// TIA Portal project "CAFERSERHAT_YAĞCI_TMR08" (V14)

(* hardware
DEVICE "S7-1200 station_1"  S7-1200 Station
   slot 0: "Rack_0"  Rack  V1.0
   slot 1: "PLC_1"  CPU 1214C DC/DC/DC  6ES7 214-1AG40-0XB0  V4.1
*)

// ===== PLC "PLC_1"  CPU 1214C DC/DC/DC =====

VAR_GLOBAL   // PLC tag table "GİRİŞ VE ÇIKIŞ ETİKETLERİ"
   "S1 NK" AT %I0.0 : Bool;
   "S5 NA" AT %I0.1 : Bool;
   "S8 NA" AT %I0.2 : Bool;
   "S8 NK" AT %I0.3 : Bool;
   "S2 NA" AT %I0.4 : Bool;
   "S2 NK" AT %I0.5 : Bool;
   "S3 NK" AT %I0.6 : Bool;
   "S3 NA" AT %I0.7 : Bool;
   "S4 NK" AT %I1.0 : Bool;
   "S4 NA" AT %I1.1 : Bool;
   "S7 NA" AT %I1.2 : Bool;
   "S7 NK" AT %I1.3 : Bool;
   "S6 NK" AT %I1.4 : Bool;
   "S6 NA" AT %I1.5 : Bool;
   "Tag_15" AT %I1.6 : Bool;
   "H2 SARI LAMBA" AT %Q0.0 : Bool;
   "H1 KIRMIZI LAMBA" AT %Q0.1 : Bool;
   "H3 SARI LAMBA" AT %Q0.2 : Bool;
   "H6 SARI LAMBA" AT %Q0.3 : Bool;
   "H5 YEŞİL LAMBA" AT %Q0.4 : Bool;
   "H7 MAVİ LAMBA" AT %Q0.5 : Bool;
   "Tag_22" AT %Q0.6 : Bool;
   "H4 YEŞİL LAMBA" AT %Q0.7 : Bool;
   "Tag_24" AT %Q1.0 : Bool;
   "Tag_25" AT %Q1.1 : Bool;
END_VAR

ORGANIZATION_BLOCK "SORU 1"   // OB1, LAD, ProgramCycle
TITLE = "Main Program Sweep (Cycle)"
{ S7_Optimized_Access := 'TRUE' }
VERSION : 0.1
   VAR_INPUT
      Initial_Call : Bool;   // Initial call of this OB
      Remanence : Bool;   // =True, if remanent data are available
   END_VAR
BEGIN

REGION Network 1
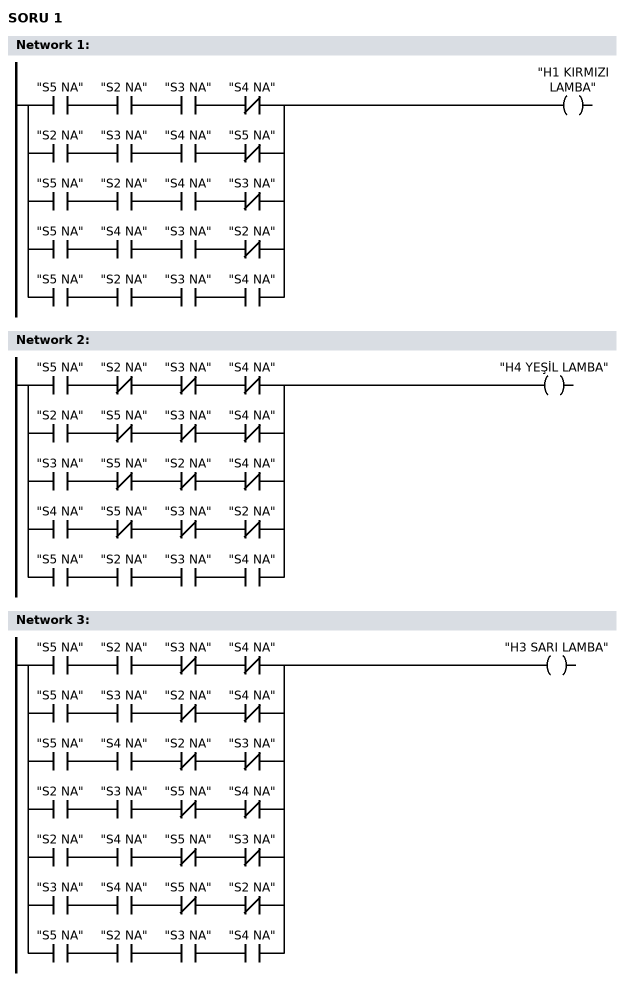
   RUNG wire#powerrail
      Contact( "S5 NA" )
      Contact( "S2 NA" )
      Contact( "S3 NA" )
      I_Contact( "S4 NA" )
      wire#w1
      Coil( "H1 KIRMIZI LAMBA" )
   END_RUNG
   RUNG wire#powerrail
      Contact( "S2 NA" )
      Contact( "S3 NA" )
      Contact( "S4 NA" )
      I_Contact( "S5 NA" )
   END_RUNG wire#w1
   RUNG wire#powerrail
      Contact( "S5 NA" )
      Contact( "S2 NA" )
      Contact( "S4 NA" )
      I_Contact( "S3 NA" )
   END_RUNG wire#w1
   RUNG wire#powerrail
      Contact( "S5 NA" )
      Contact( "S4 NA" )
      Contact( "S3 NA" )
      I_Contact( "S2 NA" )
   END_RUNG wire#w1
   RUNG wire#powerrail
      Contact( "S5 NA" )
      Contact( "S2 NA" )
      Contact( "S3 NA" )
      Contact( "S4 NA" )
   END_RUNG wire#w1
   // the same network as SCL:
   "H1 KIRMIZI LAMBA" := ("S5 NA" AND "S2 NA" AND "S3 NA" AND NOT "S4 NA") OR ("S2 NA" AND "S3 NA" AND "S4 NA" AND NOT "S5 NA") OR ("S5 NA" AND "S2 NA" AND "S4 NA" AND NOT "S3 NA") OR ("S5 NA" AND "S4 NA" AND "S3 NA" AND NOT "S2 NA") OR ("S5 NA" AND "S2 NA" AND "S3 NA" AND "S4 NA");
END_REGION

REGION Network 2
   RUNG wire#powerrail
      Contact( "S5 NA" )
      I_Contact( "S2 NA" )
      I_Contact( "S3 NA" )
      I_Contact( "S4 NA" )
      wire#w1
      Coil( "H4 YEŞİL LAMBA" )
   END_RUNG
   RUNG wire#powerrail
      Contact( "S2 NA" )
      I_Contact( "S5 NA" )
      I_Contact( "S3 NA" )
      I_Contact( "S4 NA" )
   END_RUNG wire#w1
   RUNG wire#powerrail
      Contact( "S3 NA" )
      I_Contact( "S5 NA" )
      I_Contact( "S2 NA" )
      I_Contact( "S4 NA" )
   END_RUNG wire#w1
   RUNG wire#powerrail
      Contact( "S4 NA" )
      I_Contact( "S5 NA" )
      I_Contact( "S3 NA" )
      I_Contact( "S2 NA" )
   END_RUNG wire#w1
   RUNG wire#powerrail
      Contact( "S5 NA" )
      Contact( "S2 NA" )
      Contact( "S3 NA" )
      Contact( "S4 NA" )
   END_RUNG wire#w1
   // the same network as SCL:
   "H4 YEŞİL LAMBA" := ("S5 NA" AND NOT "S2 NA" AND NOT "S3 NA" AND NOT "S4 NA") OR ("S2 NA" AND NOT "S5 NA" AND NOT "S3 NA" AND NOT "S4 NA") OR ("S3 NA" AND NOT "S5 NA" AND NOT "S2 NA" AND NOT "S4 NA") OR ("S4 NA" AND NOT "S5 NA" AND NOT "S3 NA" AND NOT "S2 NA") OR ("S5 NA" AND "S2 NA" AND "S3 NA" AND "S4 NA");
END_REGION

REGION Network 3
   RUNG wire#powerrail
      Contact( "S5 NA" )
      Contact( "S2 NA" )
      I_Contact( "S3 NA" )
      I_Contact( "S4 NA" )
      wire#w1
      Coil( "H3 SARI LAMBA" )
   END_RUNG
   RUNG wire#powerrail
      Contact( "S5 NA" )
      Contact( "S3 NA" )
      I_Contact( "S2 NA" )
      I_Contact( "S4 NA" )
   END_RUNG wire#w1
   RUNG wire#powerrail
      Contact( "S5 NA" )
      Contact( "S4 NA" )
      I_Contact( "S2 NA" )
      I_Contact( "S3 NA" )
   END_RUNG wire#w1
   RUNG wire#powerrail
      Contact( "S2 NA" )
      Contact( "S3 NA" )
      I_Contact( "S5 NA" )
      I_Contact( "S4 NA" )
   END_RUNG wire#w1
   RUNG wire#powerrail
      Contact( "S2 NA" )
      Contact( "S4 NA" )
      I_Contact( "S5 NA" )
      I_Contact( "S3 NA" )
   END_RUNG wire#w1
   RUNG wire#powerrail
      Contact( "S3 NA" )
      Contact( "S4 NA" )
      I_Contact( "S5 NA" )
      I_Contact( "S2 NA" )
   END_RUNG wire#w1
   RUNG wire#powerrail
      Contact( "S5 NA" )
      Contact( "S2 NA" )
      Contact( "S3 NA" )
      Contact( "S4 NA" )
   END_RUNG wire#w1
   // the same network as SCL:
   "H3 SARI LAMBA" := ("S5 NA" AND "S2 NA" AND NOT "S3 NA" AND NOT "S4 NA") OR ("S5 NA" AND "S3 NA" AND NOT "S2 NA" AND NOT "S4 NA") OR ("S5 NA" AND "S4 NA" AND NOT "S2 NA" AND NOT "S3 NA") OR ("S2 NA" AND "S3 NA" AND NOT "S5 NA" AND NOT "S4 NA") OR ("S2 NA" AND "S4 NA" AND NOT "S5 NA" AND NOT "S3 NA") OR ("S3 NA" AND "S4 NA" AND NOT "S5 NA" AND NOT "S2 NA") OR ("S5 NA" AND "S2 NA" AND "S3 NA" AND "S4 NA");
END_REGION
END_ORGANIZATION_BLOCK